SYSTEM TANK2_VIEWL (* 2-Tank Control System View+HMI *)
  (* Standard: 61499-1; Classification: Simulation; ApplicationDomain: Process Control *)
  (* Version 0.0, 2005-06-28, JHC, Holobloc Inc, Adapted from TANK_VIEWL *)
  DEVICE HMI : FRAME_DEVICE(BOUNDS := [100,100,150,150], GRID := [4,1])
    RESOURCE TANK1 : PANEL_RESOURCE
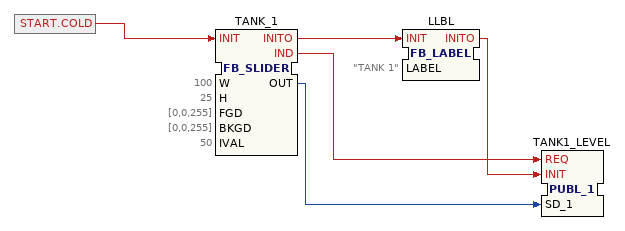
      FBS
        TANK1_LEVEL : PUBL_1;
        TANK_1 : FB_SLIDER(W := 100, H := 25, FGD := [0,0,255], BKGD := [0,0,255], IVAL := 50);
        LLBL : FB_LABEL(LABEL := "TANK 1");
      END_FBS
      EVENT_CONNECTIONS
        TANK_1.INITO TO LLBL.INIT;
        TANK_1.IND TO TANK1_LEVEL.REQ;
        START.COLD TO TANK_1.INIT;
        LLBL.INITO TO TANK1_LEVEL.INIT;
      END_CONNECTIONS
      DATA_CONNECTIONS
        TANK_1.OUT TO TANK1_LEVEL.SD_1;
      END_CONNECTIONS
    END_RESOURCE
    RESOURCE TANK2 : PANEL_RESOURCE
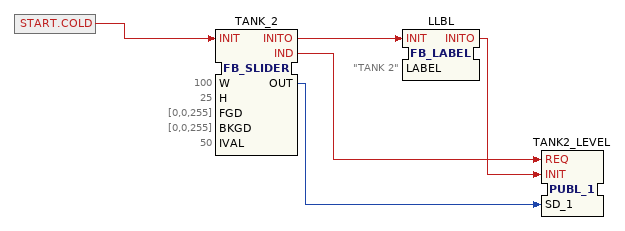
      FBS
        TANK2_LEVEL : PUBL_1;
        TANK_2 : FB_SLIDER(W := 100, H := 25, FGD := [0,0,255], BKGD := [0,0,255], IVAL := 50);
        LLBL : FB_LABEL(LABEL := "TANK 2");
      END_FBS
      EVENT_CONNECTIONS
        TANK_2.INITO TO LLBL.INIT;
        TANK_2.IND TO TANK2_LEVEL.REQ;
        START.COLD TO TANK_2.INIT;
        LLBL.INITO TO TANK2_LEVEL.INIT;
      END_CONNECTIONS
      DATA_CONNECTIONS
        TANK_2.OUT TO TANK2_LEVEL.SD_1;
      END_CONNECTIONS
    END_RESOURCE
    RESOURCE VALVE : PANEL_RESOURCE
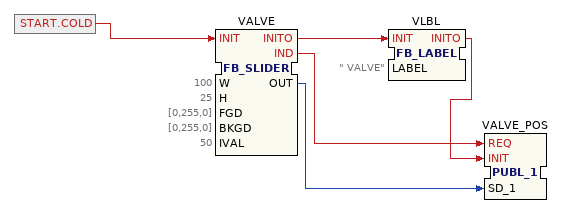
      FBS
        VALVE_POS : PUBL_1;
        VALVE : FB_SLIDER(W := 100, H := 25, FGD := [0,255,0], BKGD := [0,255,0], IVAL := 50);
        VLBL : FB_LABEL(LABEL := " VALVE");
      END_FBS
      EVENT_CONNECTIONS
        START.COLD TO VALVE.INIT;
        VALVE.INITO TO VLBL.INIT;
        VALVE.IND TO VALVE_POS.REQ;
        VLBL.INITO TO VALVE_POS.INIT;
      END_CONNECTIONS
      DATA_CONNECTIONS
        VALVE.OUT TO VALVE_POS.SD_1;
      END_CONNECTIONS
    END_RESOURCE
    RESOURCE PUMP : PANEL_RESOURCE
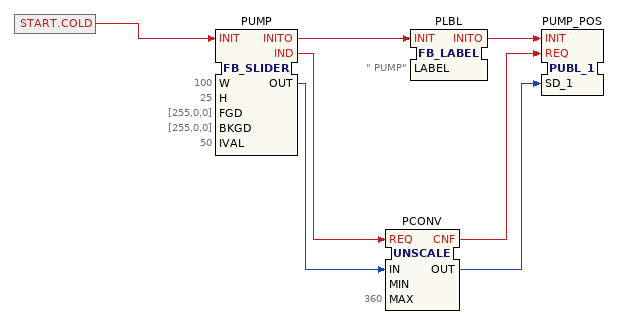
      FBS
        PUMP_POS : PUBL_1;
        PUMP : FB_SLIDER(W := 100, H := 25, FGD := [255,0,0], BKGD := [255,0,0], IVAL := 50);
        PLBL : FB_LABEL(LABEL := " PUMP");
        PCONV : UNSCALE(MAX := 360);
      END_FBS
      EVENT_CONNECTIONS
        PUMP.INITO TO PLBL.INIT;
        PLBL.INITO TO PUMP_POS.INIT;
        PUMP.IND TO PCONV.REQ;
        PCONV.CNF TO PUMP_POS.REQ;
        START.COLD TO PUMP.INIT;
      END_CONNECTIONS
      DATA_CONNECTIONS
        PUMP.OUT TO PCONV.IN;
        PCONV.OUT TO PUMP_POS.SD_1;
      END_CONNECTIONS
    END_RESOURCE
  END_DEVICE
  DEVICE VIEW : FRAME_DEVICE(BOUNDS := [250,100,238,208], GRID := [2,3])
    RESOURCE TANK1 : VIEW_PANEL(SIZE := [1,1], DIA := 75)
      FBS
        TANK : MECH_VIEW(STYLE := VSTYLE#CYLINDER, LEN := 1, DIR := 3, BKGD := [255,255,255], WKPC := [0,0,255]);
        TANK1_LEVEL : SUBL_1;
      END_FBS
      EVENT_CONNECTIONS
        TANK1_LEVEL.INITO TO TANK.INIT;
        TANK1_LEVEL.IND TO TANK.REQ;
        START.COLD TO TANK1_LEVEL.INIT;
      END_CONNECTIONS
      DATA_CONNECTIONS
        TANK1_LEVEL.RD_1 TO TANK.POS;
      END_CONNECTIONS
    END_RESOURCE
    RESOURCE VALVE : VIEW_PANEL(DIA := 75, SIZE := [1,1])
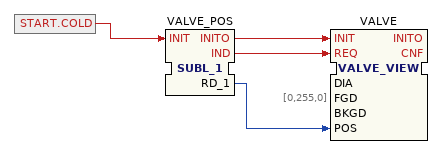
      FBS
        VALVE_POS : SUBL_1;
        VALVE : VALVE_VIEW(FGD := [0,255,0]);
      END_FBS
      EVENT_CONNECTIONS
        START.COLD TO VALVE_POS.INIT;
        VALVE_POS.INITO TO VALVE.INIT;
        VALVE_POS.IND TO VALVE.REQ;
      END_CONNECTIONS
      DATA_CONNECTIONS
        VALVE_POS.RD_1 TO VALVE.POS;
      END_CONNECTIONS
    END_RESOURCE
    RESOURCE PIPE1 : VIEW_PANEL(DIA := 38, SIZE := [2,2], VERTICAL := 1)
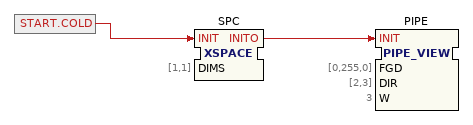
      FBS
        SPC : XSPACE(DIMS := [1,1]);
        PIPE : PIPE_VIEW(FGD := [0,255,0], DIR := [2,3], W := 3);
      END_FBS
      EVENT_CONNECTIONS
        START.COLD TO SPC.INIT;
        SPC.INITO TO PIPE.INIT;
      END_CONNECTIONS
    END_RESOURCE
    RESOURCE PIPE2 : VIEW_PANEL(DIA := 75, SIZE := [1,2])
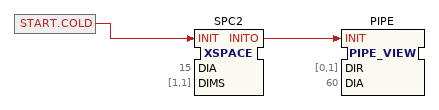
      FBS
        SPC2 : XSPACE(DIA := 15, DIMS := [1,1]);
        PIPE : PIPE_VIEW(DIR := [0,1], DIA := 60);
      END_FBS
      EVENT_CONNECTIONS
        START.COLD TO SPC2.INIT;
        SPC2.INITO TO PIPE.INIT;
      END_CONNECTIONS
    END_RESOURCE
    RESOURCE PUMP : VIEW_PANEL(DIA := 25, SIZE := [3,3], VERTICAL := 1)
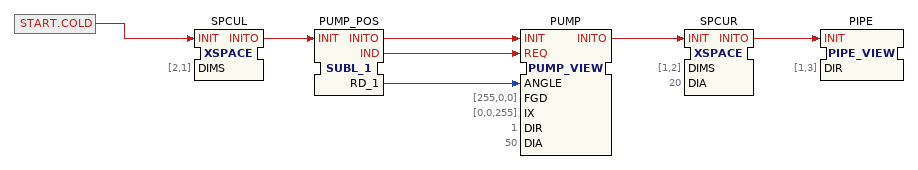
      FBS
        PUMP_POS : SUBL_1;
        SPCUL : XSPACE(DIMS := [2,1]); (* Upper Left Space *)
        PUMP : PUMP_VIEW(FGD := [255,0,0], IX := [0,0,255], DIR := 1, DIA := 50);
        PIPE : PIPE_VIEW(DIR := [1,3]);
        SPCUR : XSPACE(DIMS := [1,2], DIA := 20); (* Upper-Right Space *)
      END_FBS
      EVENT_CONNECTIONS
        PUMP_POS.INITO TO PUMP.INIT;
        PUMP_POS.IND TO PUMP.REQ;
        START.COLD TO SPCUL.INIT;
        SPCUL.INITO TO PUMP_POS.INIT;
        PUMP.INITO TO SPCUR.INIT;
        SPCUR.INITO TO PIPE.INIT;
      END_CONNECTIONS
      DATA_CONNECTIONS
        PUMP_POS.RD_1 TO PUMP.ANGLE;
      END_CONNECTIONS
    END_RESOURCE
    RESOURCE TANK2 : VIEW_PANEL(SIZE := [1,1], DIA := 75)
      FBS
        TANK : MECH_VIEW(STYLE := VSTYLE#CYLINDER, LEN := 1, DIR := 3, BKGD := [255,255,255], WKPC := [0,0,255]);
        TANK2_LEVEL : SUBL_1;
      END_FBS
      EVENT_CONNECTIONS
        TANK2_LEVEL.INITO TO TANK.INIT;
        TANK2_LEVEL.IND TO TANK.REQ;
        START.COLD TO TANK2_LEVEL.INIT;
      END_CONNECTIONS
      DATA_CONNECTIONS
        TANK2_LEVEL.RD_1 TO TANK.POS;
      END_CONNECTIONS
    END_RESOURCE
  END_DEVICE
END_SYSTEM
